// TwinCAT 3 PLC project TcOpen
// Title: TcOpen
// Company: Vortex.Library
// Author: Dustin Hullett
// ProjectVersion: 0.1.0.54
// ProgramVersion: 3.1.4023.0
// libraries:
//   Tc2_Standard, * (Beckhoff Automation GmbH)
//   Tc2_System, * (Beckhoff Automation GmbH)
//   Tc3_Module, * (Beckhoff Automation GmbH)
// project tree:
//   ComponentsBase/ fbComponent.TcPOU
//   GVLs/ IO.TcGVL
//   / PlcTask.TcTTO (not stored)
//   POUs/Cylinders/ fbCylinder.TcPOU, ICylinder.TcIO
//   POUs/ MAIN.TcPOU
//   Tasks/ eTaskState.TcDUT, fbTask.TcPOU, ITaskContainer.TcIO, ITaskStatus.TcIO (not stored)
//   Version/ Global_Version.TcGVL
//   _Tests/ MAIN_TESTS.TcPOU (not stored)
//   _Tests/Tasks/ fbTaskTests.TcPOU
// real-time tasks:
//   TASK PlcTask: cycle T#10ms, priority 20, ADS port 350

// ---- Tasks/eTaskState.TcDUT
{attribute 'qualified_only'}
{attribute 'strict'}
TYPE eTaskState :
(
	Idle := 0,
	Request := 10,
	Executing := 20,
	Error := 30,
	Done := 40
);
END_TYPE

// ---- GVLs/IO.TcGVL
{attribute 'qualified_only'}
VAR_GLOBAL 
	A1 AT %I* : ARRAY[0..7] OF BOOL;
	A2 AT %Q* : ARRAY[0..7] OF BOOL;
END_VAR

// ---- Version/Global_Version.TcGVL
{attribute 'TcGenerated'}
{attribute 'no-analysis'}
{attribute 'linkalways'}
// This function has been automatically generated from the project information.
VAR_GLOBAL CONSTANT
	{attribute 'const_non_replaced'}
	stLibVersion_TcOpen : ST_LibVersion := (iMajor := 0, iMinor := 0, iBuild := 0, iRevision := 1, nFlags := 0, sVersion := '0.0.0.1');
END_VAR

// ---- POUs/Cylinders/ICylinder.TcIO
INTERFACE ICylinder EXTENDS __System.IQueryInterface

PROPERTY AtHome : bool
GET
END_GET
END_PROPERTY

PROPERTY AtWork : bool
GET
END_GET
END_PROPERTY

METHOD MoveToHome : ITask
END_METHOD

METHOD MoveToWork : ITask
END_METHOD

END_INTERFACE

// ---- Tasks/ITaskContainer.TcIO
INTERFACE ITaskContainer

PROPERTY Lock : INT
GET
END_GET
SET
END_SET
END_PROPERTY

END_INTERFACE

// ---- ComponentsBase/fbComponent.TcPOU
FUNCTION_BLOCK ABSTRACT fbComponent IMPLEMENTS IComponent
VAR	
	{attribute addProperty Name "Components' message"}
	{attribute clr [ReadOnly()]}
	_message : STRING(255);
	{attribute 'hide'}
	_lock : INT;		
END_VAR

METHOD PROTECTED Info
VAR_INPUT
	inMessage : STRING(255);
END_VAR
_message := inMessage;
END_METHOD

PROPERTY Lock : INT
GET
Lock := _lock;
END_GET
SET
_lock := Lock;
END_SET
END_PROPERTY

METHOD PUBLIC Manual
THIS^.ManualControl();
END_METHOD

METHOD PROTECTED ABSTRACT ManualControl
END_METHOD

END_FUNCTION_BLOCK

// ---- POUs/Cylinders/fbCylinder.TcPOU
FUNCTION_BLOCK fbCylinder EXTENDS fbComponent IMPLEMENTS ICylinder
VAR_INPUT
	(*~
		<docu>
			<summary>
				Home position sensor.
			</summary>	
		</docu>
	~*)
	{attribute wpf [Container(Layout.UniformGrid)]}
	{attribute wpf [Group(Layout.GroupBox, "Inputs")]}	
	{attribute addProperty Name "Home position sensor"}
	inAtHomePos : BOOL;
	(*~
		<docu>
			<summary>
				Working position sensor.
			</summary>	
		</docu>
	~*) 
	{attribute addProperty Name "Work position sensor"}
	inAtWorkPos : BOOL; 
END_VAR
VAR_OUTPUT
	(*~
		<docu>
			<summary>
				Move to working home position signal.
			</summary>	
		</docu>
	~*)
	{attribute wpf [Container(Layout.UniformGrid)]}
	{attribute wpf [Group(Layout.GroupBox, "Outputs")]}	
	{attribute addProperty Name "Move to home position actuator"}
	outToHomePos : BOOL;
	(*~
		<docu>
			<summary>
				Move to working posistion signal.
			</summary>	
		</docu>
	~*)
	{attribute addProperty Name "Move to work position actuator"}
	outToWorkPos : BOOL;
END_VAR

VAR	
	{attribute wpf [Container(Layout.UniformGrid)]}
	{attribute addProperty Name "Request move to Home position"}	
	_moveHomeTask : fbTask(THIS^);
	{attribute addProperty Name "Request move to Work position"}
	_moveWorkTask : fbTask(THIS^);
	{attribute addProperty Name "Request Stop"}
	_stopTask : fbTask(THIS^);
END_VAR

IF(_moveHomeTask.Execute(1)) THEN
	outToHomePos := TRUE;
	outToWorkPos := FALSE; 		
	_moveHomeTask.DoneWhen(inAtHomePos);			
END_IF

IF(_moveWorkTask.Execute(2)) THEN
	outToWorkPos := TRUE; 
	outToHomePos := FALSE;
	_moveWorkTask.DoneWhen(inAtWorkPos);
END_IF;	 

IF(_stopTask.Execute(0)) THEN	
	outToWorkPos := FALSE; 
	outToHomePos := FALSE;
	_moveWorkTask.Reset();
	_moveHomeTask.Reset();
	_stopTask.Reset();
	_stopTask.DoneWhen(TRUE);	
END_IF

{attribute 'TcRpcEnable'}
METHOD INTERNAL _MoveToHomeTest : BOOL
_MoveToHomeTest := MoveToHome().Done;
END_METHOD

{attribute 'TcRpcEnable'}
METHOD INTERNAL _MoveToWorkTest : BOOL
_MoveToWorkTest := MoveToWork().Done;
END_METHOD

{attribute 'TcRpcEnable'}
METHOD INTERNAL _StopTest : BOOL
_StopTest := Stop().Done;
END_METHOD

PROPERTY AtHome : bool
GET
AtHome := inAtHomePos;
END_GET
END_PROPERTY

PROPERTY AtWork : bool
GET
AtWork := inAtWorkPos;
END_GET
END_PROPERTY

METHOD PROTECTED  ManualControl
END_METHOD

(*~
	<docu>
		<summary>
			Moves the piston into home position.
		</summary>
		<returns>True when home position sensor is reached.</returns>
	</docu>
~*)
METHOD MoveToHome : ITaskStatus
THIS^._moveHomeTask.Invoke();
MoveToHome := THIS^._moveHomeTask;
END_METHOD

(*~
	<docu>
		<summary>
			Moves the piston into working position.
		</summary>
		<returns>True when working position sensor is reached.</returns>
	</docu>
~*)
METHOD MoveToWork : ITaskStatus
THIS^._moveWorkTask.Invoke();
MoveToWork := THIS^._moveWorkTask;
END_METHOD

METHOD Stop : REFERENCE TO fbTask
_stopTask.Invoke();
Stop REF= _stopTask;
END_METHOD

END_FUNCTION_BLOCK

// ---- Tasks/fbTask.TcPOU
FUNCTION_BLOCK fbTask IMPLEMENTS ITaskStatus
VAR
	_taskState : eTaskState;
	_ipComponent : ITaskContainer;	
END_VAR

METHOD Abort
THIS^.Reset();
END_METHOD

PROPERTY Busy : BOOL
GET
Busy := THIS^._taskState = eTaskState.Executing;
END_GET
END_PROPERTY

PROPERTY Done : BOOL
GET
Done := THIS^._taskState = eTaskState.Done;

IF(Done) THEN
	THIS^._taskState := eTaskState.Idle;
END_IF
END_GET
END_PROPERTY

METHOD DoneWhen 
VAR_INPUT
	Condition : BOOL;
END_VAR
IF (Condition) THEN
	THIS^._taskState := eTaskState.Done;
	THIS^._ipComponent.Lock := 0;			
END_IF;
END_METHOD

PROPERTY Error : BOOL
GET
Error := THIS^._taskState = eTaskState.Error;
END_GET
END_PROPERTY

METHOD Execute : BOOL
VAR_INPUT
	key : INT := 0;
END_VAR
IF(THIS^._taskState = eTaskState.Request 
  AND_THEN (THIS^._ipComponent.Lock = 0 
  OR THIS^._ipComponent.Lock = key)) 
  THEN
	THIS^._taskState := eTaskState.Executing;
	THIS^._ipComponent.Lock := key;
END_IF;
	
Execute := (THIS^._taskState = eTaskState.Executing);
END_METHOD

METHOD PUBLIC FB_init : BOOL
VAR_INPUT
	bInitRetains : BOOL; // if TRUE, the retain variables are initialized (warm start / cold start)
	bInCopyCode : BOOL;  // if TRUE, the instance afterwards gets moved into the copy code (online change)
	component : ITaskContainer;
END_VAR
_ipComponent := component;
END_METHOD

METHOD Invoke
IF(THIS^._taskState < eTaskState.Error) THEN
	THIS^._taskState := eTaskState.Request;
END_IF;
END_METHOD

METHOD Reset
VAR_INPUT
END_VAR
THIS^._taskState := eTaskState.Idle;
END_METHOD

METHOD ThrowWhen
VAR_INPUT
	condition : BOOL;
END_VAR
IF (condition) THEN
	THIS^._taskState := eTaskState.Error;
END_IF
END_METHOD

END_FUNCTION_BLOCK

// ---- POUs/MAIN.TcPOU
PROGRAM MAIN
VAR	
	{attribute wpf [Container(Layout.Stack)]}	
	{attribute addProperty Name "WPF cyclinder"}
	_wpfCyclinder : fbCylinder;	
	{attribute wpf [Container(Layout.Stack)]}	
	{attribute addProperty Name "WPF cyclinder 1"}
	_wpfCyclinder_1 : fbCylinder;
	{attribute wpf [Container(Layout.Stack)]}	
	{attribute addProperty Name "WPF cyclinder 2"}
	_wpfCyclinder_2 : fbCylinder;
	{attribute wpf [Container(Layout.Stack)]}	
	{attribute addProperty Name "WPF cyclinder 3"}
	_wpfCyclinder_3 : fbCylinder;	
END_VAR

_wpfCyclinder(inAtHomePos:=IO.A1[0] , inAtWorkPos:=IO.A1[1] , outToHomePos=> IO.A2[0], outToWorkPos=>IO.A2[1]);

_wpfCyclinder.Manual();
_wpfCyclinder_1.Manual();
_wpfCyclinder_2.Manual();
_wpfCyclinder_3.Manual();

END_PROGRAM

// ---- _Tests/Tasks/fbTaskTests.TcPOU
FUNCTION_BLOCK INTERNAL fbTaskTests EXTENDS fbComponent
VAR			
	_task_index : UINT;
	_tasks : ARRAY[0..NUMBER_OF_TASKS] OF fbTask(THIS^); 
	_task_lock_group : ARRAY[0..NUMBER_OF_TASKS] OF UINT;
	_task_done_condition : ARRAY[0..NUMBER_OF_TASKS] OF BOOL;	
	_task_fail_condition : ARRAY[0..NUMBER_OF_TASKS] OF BOOL; 	
END_VAR

VAR CONSTANT
	NUMBER_OF_TASKS : UINT := 4;
END_VAR

_task_index := 0;
IF(_tasks[_task_index].Execute(_task_lock_group[_task_index])) THEN
	_tasks[_task_index].DoneWhen(_task_done_condition[_task_index]);
	_tasks[_task_index].ThrowWhen(_task_fail_condition[_task_index]);
END_IF


_task_index := _task_index + 1;
IF(_tasks[_task_index].Execute(_task_lock_group[_task_index])) THEN
	_tasks[_task_index].DoneWhen(_task_done_condition[_task_index]);
	_tasks[_task_index].ThrowWhen(_task_fail_condition[_task_index]);
END_IF

_task_index := _task_index + 1;
IF(_tasks[_task_index].Execute(_task_lock_group[_task_index])) THEN
	_tasks[_task_index].DoneWhen(_task_done_condition[_task_index]);
	_tasks[_task_index].ThrowWhen(_task_fail_condition[_task_index]);
END_IF

_task_index := _task_index + 1;
IF(_tasks[_task_index].Execute(_task_lock_group[_task_index])) THEN
	_tasks[_task_index].DoneWhen(_task_done_condition[_task_index]);
	_tasks[_task_index].ThrowWhen(_task_fail_condition[_task_index]);
END_IF

_task_index := _task_index + 1;
IF(_tasks[_task_index].Execute(_task_lock_group[_task_index])) THEN
	_tasks[_task_index].DoneWhen(_task_done_condition[_task_index]);
	_tasks[_task_index].ThrowWhen(_task_fail_condition[_task_index]);
END_IF

{attribute 'TcRpcEnable'}
METHOD AbortTest
VAR_INPUT
	taskIndex : UINT;
END_VAR
THIS^._tasks[taskIndex].Reset();
END_METHOD

{attribute 'TcRpcEnable'}
METHOD GetBusyTest : BOOL;
VAR_INPUT
	taskIndex : UINT;
END_VAR
GetBusyTest := THIS^._tasks[taskIndex].Busy;
END_METHOD

{attribute 'TcRpcEnable'}
METHOD GetDoneTest : BOOL;
VAR_INPUT
	taskIndex : UINT;
END_VAR
GetDoneTest := THIS^._tasks[taskIndex].Done;
END_METHOD

{attribute 'TcRpcEnable'}
METHOD GetErrorTest : BOOL;
VAR_INPUT
	taskIndex : UINT;
END_VAR
GetErrorTest := THIS^._tasks[taskIndex].Error;
END_METHOD

METHOD InvokeTask : ITaskStatus
VAR_INPUT
	taskIndex : UINT;
END_VAR
THIS^._tasks[taskIndex].Invoke();
InvokeTask := THIS^._tasks[taskIndex];
END_METHOD

{attribute 'TcRpcEnable'}
METHOD InvokeTaskTest
VAR_INPUT
	taskIndex : UINT;
END_VAR
InvokeTask(taskIndex);
END_METHOD

{attribute 'TcRpcEnable'}
METHOD INTERNAL InvokeTaskTests_with_done : BOOL
VAR_INPUT
	taskIndex : UINT;
END_VAR
InvokeTaskTests_with_done := InvokeTask(taskIndex).Done;
END_METHOD

METHOD PROTECTED  ManualControl
END_METHOD

{attribute 'TcRpcEnable'}
METHOD ResetComponent
VAR_INPUT
END_VAR
THIS^.Lock := 0;
END_METHOD

{attribute 'TcRpcEnable'}
METHOD ResetTask
VAR_INPUT
	taskIndex : UINT;
END_VAR
THIS^._tasks[taskIndex].Reset();
END_METHOD

END_FUNCTION_BLOCK
